// TIA Portal V20 export
TYPE "ConveyorParameters"
// stored: Access Published, Namespace LineA1
   STRUCT
      StartUpTime : Time := T#0S;
      SensorFilterTime : Array[1..2] of Time;
      SensorBlockageTime : Time := T#5S;
      EnergySaveTime : Time := T#3s;
      ConvOccTime : Time := T#1000ms;
   END_STRUCT;
   // SensorFilterTime[1..2] := T#10ms;
END_TYPE
